// TIA Portal V19 export
DATA_BLOCK "HmiInterface"   // DB45
// stored: Access Published, MemoryReserve 100, Namespace Unit3.EM1
   VAR
      em : "LAF_typeEmInterface";
      jobs : "LAF_typeJobsInterface";
      sequence : "LAF_typeSequenceInterface";
      cm1SignalTm { S7_SetPoint := 'True'} : "EXCHANGETRAY_typeNgConveyorIoSignalInterface";
      cm2AxisControl : "LBC_typeAxisSimpleControlInterface_1";
      cm3NgStrapPositionDetection : "LEXCHANGETRAY_typeNgStrapInterface";
      cm4FrButton { S7_SetPoint := 'True'} : "EXCHANGETRAY_typeFrButtonInterface";
      em1Parameters { S7_SetPoint := 'True'} : "LAF_typeNgConveyorEm1ParametersInterface";
   END_VAR
BEGIN
   cm1SignalTm.commands.ngStrapSignal := TRUE;
   cm1SignalTm.commands.ngSafeDoorSignal := true;
END_DATA_BLOCK
